// Function block with properties demonstrating TwinCAT 3 OOP features

FUNCTION_BLOCK FB_WithProperties

VAR
    nInternal : INT := 0;
    fInternalValue : REAL := 0.0;
    sInternalName : STRING(50) := '';
END_VAR

// Main execution - no-op for property demo

// Property: Value
// Gets or sets the internal integer value

PROPERTY Value : INT
GET
// Getter for Value property

VAR
END_VAR
Value := nInternal;
END_GET
SET
// Setter for Value property

VAR
END_VAR
nInternal := Value;
END_SET
END_PROPERTY

// Property: ReadOnlyStatus
// Read-only property returning calculated status

PROPERTY ReadOnlyStatus : INT
GET
// Getter for ReadOnlyStatus property

VAR
    nCalcStatus : INT;
END_VAR
nCalcStatus := nInternal * 2;
ReadOnlyStatus := nCalcStatus;
END_GET
END_PROPERTY

// Property: Name
// Gets or sets the internal name string

PROPERTY Name : STRING(50)
GET
// Getter for Name property

VAR
END_VAR
Name := sInternalName;
END_GET
SET
// Setter for Name property

VAR
END_VAR
sInternalName := Name;
END_SET
END_PROPERTY

END_FUNCTION_BLOCK

(* stored: Version 1.1.0.1
   POU FB_WithProperties: Id {bbbbbbbb-cccc-dddd-eeee-ffffffffffff}, SpecialFunc None
   Property Value: Id {44444444-5555-6666-7777-888888888888}
   Get Get: Id {44444444-5555-6666-7777-888888888889}
   Set Set: Id {44444444-5555-6666-7777-88888888888a}
   Property ReadOnlyStatus: Id {55555555-6666-7777-8888-999999999999}
   Get Get: Id {55555555-6666-7777-8888-99999999999a}
   Property Name: Id {66666666-7777-8888-9999-aaaaaaaaaaaa}
   Get Get: Id {66666666-7777-8888-9999-aaaaaaaaaa0b}
   Set Set: Id {66666666-7777-8888-9999-aaaaaaaaaa0c} *)
